FUNCTION_BLOCK FB_Motion
VAR_INPUT
END_VAR
VAR_OUTPUT
END_VAR
VAR
	MCPower: MC_Power;
	MCMoveAbs: MC_MoveAbsolute;
	MCStop: MC_Stop;
	MCReset: MC_Reset;
END_VAR

VAR_IN_OUT
	Axis	:	AXIS_REF;
	StAxis	:	ST_Axis;
END_VAR

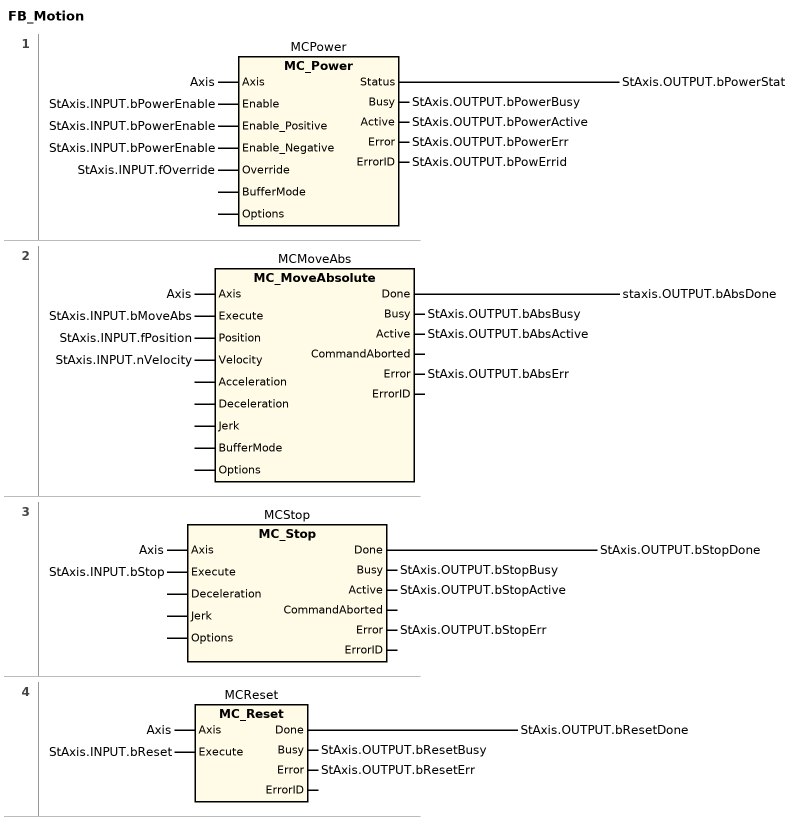
// NETWORK 1
MCPower(
    Axis := Axis,
    Enable := StAxis.INPUT.bPowerEnable,
    Enable_Positive := StAxis.INPUT.bPowerEnable,
    Enable_Negative := StAxis.INPUT.bPowerEnable,
    Override := StAxis.INPUT.fOverride,
    Busy => StAxis.OUTPUT.bPowerBusy,
    Active => StAxis.OUTPUT.bPowerActive,
    Error => StAxis.OUTPUT.bPowerErr,
    ErrorID => StAxis.OUTPUT.bPowErrid); // MC_Power
StAxis.OUTPUT.bPowerStat := MCPower.Status;

// NETWORK 2
MCMoveAbs(
    Axis := Axis,
    Execute := StAxis.INPUT.bMoveAbs,
    Position := StAxis.INPUT.fPosition,
    Velocity := StAxis.INPUT.nVelocity,
    Busy => StAxis.OUTPUT.bAbsBusy,
    Active => StAxis.OUTPUT.bAbsActive,
    Error => StAxis.OUTPUT.bAbsErr); // MC_MoveAbsolute
staxis.OUTPUT.bAbsDone := MCMoveAbs.Done;

// NETWORK 3
MCStop(
    Axis := Axis,
    Execute := StAxis.INPUT.bStop,
    Busy => StAxis.OUTPUT.bStopBusy,
    Active => StAxis.OUTPUT.bStopActive,
    Error => StAxis.OUTPUT.bStopErr); // MC_Stop
StAxis.OUTPUT.bStopDone := MCStop.Done;

// NETWORK 4
MCReset(
    Axis := Axis,
    Execute := StAxis.INPUT.bReset,
    Busy => StAxis.OUTPUT.bResetBusy,
    Error => StAxis.OUTPUT.bResetErr); // MC_Reset
StAxis.OUTPUT.bResetDone := MCReset.Done;

END_FUNCTION_BLOCK

(* stored: Version 1.1.0.1, ProductVersion 3.1.4022.18
   POU FB_Motion: Id {4e398971-6192-4d27-a7cc-c245b8793513}, SpecialFunc None *)
